TYPE "Check"
VERSION : 0.1
   STRUCT
      Mode : Bool;
      DataClear : Bool;
      Code : Array[0..10] of String[48];
      Choice1 : Bool;
      Choice2 : Bool;
      Choice3 : Bool;
      Choice4 : Bool;
      Choice5 : Bool;
      Choice6 : Bool;
      Choice7 : Bool;
      Choice8 : Bool;
      TotalResult : Array[0..10] of Int;
      OP2Result : Array[0..10] of Int;
      OP5Result : Array[0..10] of Int;
      AllResult : Int;
      LoadInx : Int;
   END_STRUCT;

END_TYPE

